// TIA Portal project "Project_teste" (V17)

(* hardware
DEVICE "S7-1200 station_1"  S7-1200 Station
   slot 0: "Rack_0"  S7-1200 Rack  Rack  V1.0
   slot 1: "PLC_1"  CPU 1214C DC/DC/DC  6ES7 214-1AG40-0XB0  V4.4
*)

// ===== PLC "PLC_1"  CPU 1214C DC/DC/DC =====

VAR_GLOBAL   // PLC tag table "Default tag table"
   "liga" AT %I0.0 : Bool;
   "velocidade" AT %MW2 : UInt;
   "velocidade_motor" AT %MW4 : Word;
   "corrente_motor" AT %MW6 : Word;
   "falha_motor" AT %MW8 : Word;
   "troca_ref" AT %I0.1 : Bool;
END_VAR

TYPE "driver_config"
   STRUCT
      MB_client : TCON_IP_v4;
   END_STRUCT;
   // MB_client.InterfaceId := 64;
   // MB_client.ID := 1;
   // MB_client.ConnectionType := 11;
   // MB_client.ActiveEstablished := true;
   // MB_client.RemotePort := 502;
   // MB_client.LocalPort := 502;
END_TYPE

TYPE "driver_comunic"
   STRUCT
      parametros : Array[0..3] of UDInt;
      leitura_escrita : Array[0..3] of Bool;
      dado_leitura : Array[0..3] of Word;
      dado_escrita : Array[0..3] of Word;
      trigger : Array[0..3] of Bool;
   END_STRUCT;
END_TYPE

DATA_BLOCK "configuracao"   // DB1
{ S7_Optimized_Access := 'TRUE' }
VERSION : 0.1
BEGIN
   MB_client.RemoteAddress.ADDR[1] := 172;
   MB_client.RemoteAddress.ADDR[2] := 16;
   MB_client.RemoteAddress.ADDR[3] := 80;
   MB_client.RemoteAddress.ADDR[4] := 30;
END_DATA_BLOCK

DATA_BLOCK "comunicacao"   // DB2
{ S7_Optimized_Access := 'TRUE' }
VERSION : 0.1
BEGIN
END_DATA_BLOCK

DATA_BLOCK "Driver_CFW500_DB"   // DB4
{ S7_Optimized_Access := 'TRUE' }
VERSION : 0.1
// stored: InstanceOfName Driver_CFW500
"Driver_CFW500"
BEGIN
END_DATA_BLOCK

FUNCTION_BLOCK "transicao_estados"   // FB1, SCL
{ S7_Optimized_Access := 'FALSE' }
VERSION : 0.1
   VAR_INPUT
      liga : Bool;
      ref_velocidade : UInt;
      rampa_aceleracao : UInt;
      rampa_desaceleracao : UInt;
   END_VAR
BEGIN
   CASE "Driver_CFW500_DB".estado OF
       0:
           IF NOT "Driver_CFW500_DB".saidas_atualizadas THEN
               "Driver_CFW500_DB".estado := 1;
           END_IF;
       1:
           IF "Driver_CFW500_DB".saidas_atualizadas THEN
               "Driver_CFW500_DB".estado := 10;
           END_IF;
       10:  
           IF #liga <> "Driver_CFW500_DB".ligar_old THEN
               "Driver_CFW500_DB".estado := 100;
           ELSE
               "Driver_CFW500_DB".estado := 11;
           END_IF;
       11:  
           IF #ref_velocidade <> "Driver_CFW500_DB".ref_velocidade_old THEN
               "Driver_CFW500_DB".estado := 101;
           ELSE
               "Driver_CFW500_DB".estado := 12;
           END_IF;
       12:
           IF #rampa_aceleracao <> "Driver_CFW500_DB".rampa_aceleracao_old THEN
               "Driver_CFW500_DB".estado := 102;
           ELSE
               "Driver_CFW500_DB".estado := 13;
           END_IF;
       13:
           IF #rampa_desaceleracao <> "Driver_CFW500_DB".rampa_desaceleracao_old THEN
               "Driver_CFW500_DB".estado := 103;
           ELSE
               "Driver_CFW500_DB".estado := 49;
           END_IF;
       49:
           IF NOT "Driver_CFW500_DB".param_var_atualizados THEN
               "Driver_CFW500_DB".estado := 50;
           END_IF;
       50:
           IF "Driver_CFW500_DB".param_var_atualizados THEN
               "Driver_CFW500_DB".estado := 0;
           END_IF;
       100:
           IF #liga = "Driver_CFW500_DB".ligar_old THEN
               "Driver_CFW500_DB".estado := 49;
           END_IF;
       101:
           IF #ref_velocidade = "Driver_CFW500_DB".ref_velocidade_old THEN
               "Driver_CFW500_DB".estado := 49;
           END_IF;
       102:
           IF #rampa_aceleracao = "Driver_CFW500_DB".rampa_aceleracao_old THEN
               "Driver_CFW500_DB".estado := 49;
           END_IF;
       103:
           IF #rampa_desaceleracao = "Driver_CFW500_DB".rampa_desaceleracao_old THEN
               "Driver_CFW500_DB".estado := 49;
           END_IF;
   END_CASE;
END_FUNCTION_BLOCK

FUNCTION_BLOCK "escrever_parametro"   // FB2, SCL
{ S7_Optimized_Access := 'FALSE' }
VERSION : 0.1
   VAR_INPUT
      parametro : UDInt;
      dado : Word;
      escrever : Bool;
   END_VAR
   VAR_OUTPUT
      escrito : Bool;
   END_VAR
   VAR
      flag_start : Bool;
   END_VAR
BEGIN
   IF #escrever AND
      NOT #flag_start AND
      NOT "Driver_CFW500_DB".disconnect AND
      NOT "Driver_CFW500_DB".busy THEN

       #escrito := 0;

       // Define modo de escrita
       "Driver_CFW500_DB".mode := 1;

       // Define comprimento da escrita
       "Driver_CFW500_DB".data_len := 1;

       // Define endereço para escrita
       "Driver_CFW500_DB".data_addr := #parametro + 40001;

       // Define dado para escrita
       "Driver_CFW500_DB".data_ptr[0] := #dado;

       // Gera pulso para disparar requisição de escrita
       "Driver_CFW500_DB".req := 1;

       #flag_start := TRUE;

   ELSIF #flag_start AND "Driver_CFW500_DB".busy THEN
       "Driver_CFW500_DB".req := FALSE;

   ELSIF #flag_start AND
      ("Driver_CFW500_DB".done OR "Driver_CFW500_DB".error) THEN
      #flag_start := FALSE;
      #escrito := TRUE;

   END_IF;
END_FUNCTION_BLOCK

FUNCTION_BLOCK "ler_parametro"   // FB3, SCL
{ S7_Optimized_Access := 'FALSE' }
VERSION : 0.1
   VAR_INPUT
      parametro : UDInt;
      ler : Bool;
   END_VAR
   VAR_OUTPUT
      dado : Word;
      lido : Bool;
   END_VAR
   VAR
      flag_start : Bool;
   END_VAR
BEGIN
   IF #ler AND
       NOT #flag_start AND
       NOT "Driver_CFW500_DB".disconnect AND
       NOT "Driver_CFW500_DB".busy THEN

       //    "Driver_CFW500_DB".data_ptr[0] := 0;
       //    #dado := 0;
       #lido := FALSE;

       // Define modo de leitura
       "Driver_CFW500_DB".mode := 0;

       // Define comprimento da leitura
       "Driver_CFW500_DB".data_len := 1;

       // Define endereço para leitura
       "Driver_CFW500_DB".data_addr := #parametro + 40001;

       // Gera pulso para disparar requisição de leitura
       "Driver_CFW500_DB".req := 1;

       #flag_start := TRUE;

   ELSIF #flag_start AND "Driver_CFW500_DB".busy THEN
       "Driver_CFW500_DB".req := FALSE;

   ELSIF #flag_start AND
         NOT "Driver_CFW500_DB".req AND
         ("Driver_CFW500_DB".done OR "Driver_CFW500_DB".error) THEN

       #flag_start := FALSE;
       #dado := "Driver_CFW500_DB".data_ptr[0];
       #lido := TRUE;

   END_IF;
END_FUNCTION_BLOCK

FUNCTION_BLOCK "acoes_estado"   // FB4, LAD
{ S7_Optimized_Access := 'FALSE' }
VERSION : 0.1
   VAR_INPUT
      ligar : Bool;
      ref_vel : Word;
      rampa_acel : Word;
      rampa_desacel : Word;
   END_VAR
   VAR_OUTPUT
      velocidade : Word;
      corrente : Word;
      falha : Word;
   END_VAR
   VAR
      aux0 : Bool;
      aux1 : Bool;
      aux2 : Bool;
      aux3 : Bool;
      aux4 : Bool;
      aux5 : Bool;
      aux6 : Bool;
      aux7 : Bool;
      aux10 : Bool;
      aux11 : Bool;
      aux12 : Bool;
      aux13 : Bool;
      aux20 : Bool;
      aux21 : Bool;
      aux22 : Bool;
      aux23 : Bool;
      aux30 : Bool;
      aux31 : Bool;
      aux32 : Bool;
      aux33 : Bool;
      aux100 : Bool;
      aux101 : Bool;
      aux102 : Bool;
      aux103 : Bool;
      aux104 : Bool;
      aux105 : Bool;
      aux106 : Bool;
      aux107 : Bool;
      aux200 : Bool;
      aux201 : Bool;
      aux202 : Bool;
      aux203 : Bool;
      aux204 : Bool;
      aux205 : Bool;
      aux206 : Bool;
      aux207 : Bool;
      aux208 : Bool;
      aux209 : Bool;
      aux210 : Bool;
      aux211 : Bool;
      atualizar_p0 : Bool;
      atualizar_p1 : Bool;
      atualizar_p2 : Bool;
      atualizar_p3 : Bool;
      ler_vel : "ler_parametro";
      ler_cor : "ler_parametro";
      ler_falha : "ler_parametro";
      escrever_liga : "escrever_parametro";
      escrever_desliga : "escrever_parametro";
      escrever_ref : "escrever_parametro";
      escrever_acel : "escrever_parametro";
      escrever_desacel : "escrever_parametro";
      est_50 : "estado 50";
      temporiza : IEC_TIMER;
   END_VAR
   VAR_TEMP   // added for the SCL form of the ladder/FBD networks
      _w1 : Bool;
      _w2 : Bool;
      _w3 : Bool;
      _w4 : Bool;
      _w5 : Bool;
   END_VAR
BEGIN

REGION Network 1: Estado 0
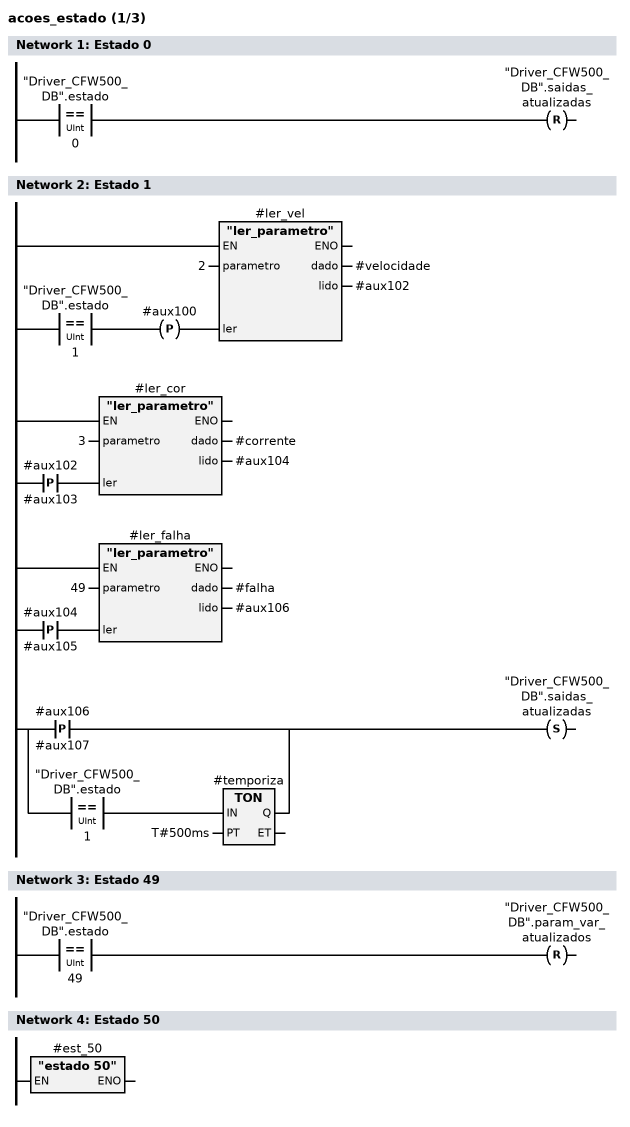
   RUNG wire#powerrail
      { S7_Templates := "SrcType := UInt" } EQ_Contact(in1 := "Driver_CFW500_DB".estado, in2 := 0)
      R_Coil( "Driver_CFW500_DB".saidas_atualizadas )
   END_RUNG
   // the same network as SCL:
   IF "Driver_CFW500_DB".estado = 0 THEN "Driver_CFW500_DB".saidas_atualizadas := FALSE; END_IF;
END_REGION

REGION Network 2: Estado 1
   #_w1 := "Driver_CFW500_DB".estado = 1;
   #_w2 := #_w1 AND NOT #aux100;   // rising edge
   #aux100 := #_w1;
   #ler_vel(parametro := 2, ler := #_w2, dado => #velocidade, lido => #aux102);   // "ler_parametro"
   #_w3 := #aux102 AND NOT #aux103;   // rising edge of #aux102
   #aux103 := #aux102;
   #ler_cor(parametro := 3, ler := #_w3, dado => #corrente, lido => #aux104);   // "ler_parametro"
   #_w4 := #aux104 AND NOT #aux105;   // rising edge of #aux104
   #aux105 := #aux104;
   #ler_falha(parametro := 49, ler := #_w4, dado => #falha, lido => #aux106);   // "ler_parametro"
   #_w5 := #aux106 AND NOT #aux107;   // rising edge of #aux106
   #aux107 := #aux106;
   #temporiza.TON(IN := "Driver_CFW500_DB".estado = 1, PT := T#500ms);
   IF #_w5 OR #temporiza.Q THEN "Driver_CFW500_DB".saidas_atualizadas := TRUE; END_IF;
END_REGION

REGION Network 3: Estado 49
   RUNG wire#powerrail
      { S7_Templates := "SrcType := UInt" } EQ_Contact(in1 := "Driver_CFW500_DB".estado, in2 := 49)
      R_Coil( "Driver_CFW500_DB".param_var_atualizados )
   END_RUNG
   // the same network as SCL:
   IF "Driver_CFW500_DB".estado = 49 THEN "Driver_CFW500_DB".param_var_atualizados := FALSE; END_IF;
END_REGION

REGION Network 4: Estado 50
   RUNG wire#powerrail
      #est_50()
   END_RUNG
   // the same network as SCL:
   #est_50();   // "estado 50"
END_REGION

REGION Network 5: Estado 100
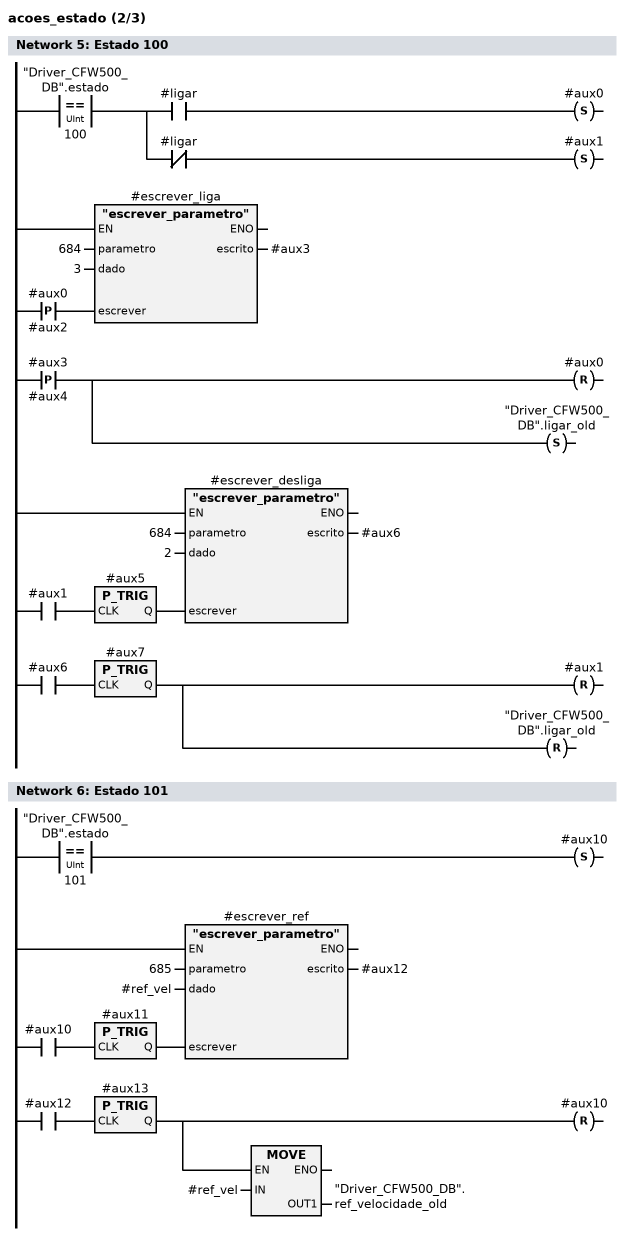
   RUNG wire#powerrail
      { S7_Templates := "SrcType := UInt" } EQ_Contact(in1 := "Driver_CFW500_DB".estado, in2 := 100)
      wire#w1
      Contact( #ligar )
      S_Coil( #aux0 )
   END_RUNG
   RUNG wire#w1
      I_Contact( #ligar )
      S_Coil( #aux1 )
   END_RUNG
   RUNG wire#powerrail
      #escrever_liga(escrever := wire#w2, parametro := 684, dado := 3, escrito => #aux3)
   END_RUNG
   RUNG wire#powerrail
      P_Contact(operand := #aux0, bit := #aux2)
   END_RUNG wire#w2
   RUNG wire#powerrail
      P_Contact(operand := #aux3, bit := #aux4)
      wire#w3
      R_Coil( #aux0 )
   END_RUNG
   RUNG wire#w3
      S_Coil( "Driver_CFW500_DB".ligar_old )
   END_RUNG
   RUNG wire#powerrail
      #escrever_desliga(escrever := wire#w4, parametro := 684, dado := 2, escrito => #aux6)
   END_RUNG
   RUNG wire#powerrail
      Contact( #aux1 )
      P_Trig( #aux5 )
   END_RUNG wire#w4
   RUNG wire#powerrail
      Contact( #aux6 )
      P_Trig( #aux7 )
      wire#w5
      R_Coil( #aux1 )
   END_RUNG
   RUNG wire#w5
      R_Coil( "Driver_CFW500_DB".ligar_old )
   END_RUNG
   // the same network as SCL:
   #_w1 := "Driver_CFW500_DB".estado = 100;
   IF #_w1 AND #ligar THEN #aux0 := TRUE; END_IF;
   IF #_w1 AND NOT #ligar THEN #aux1 := TRUE; END_IF;
   #_w2 := #aux0 AND NOT #aux2;   // rising edge of #aux0
   #aux2 := #aux0;
   #escrever_liga(parametro := 684, dado := 3, escrever := #_w2, escrito => #aux3);   // "escrever_parametro"
   #_w3 := #aux3 AND NOT #aux4;   // rising edge of #aux3
   #aux4 := #aux3;
   IF #_w3 THEN
       #aux0 := FALSE;
       "Driver_CFW500_DB".ligar_old := TRUE;
   END_IF;
   #_w4 := #aux1 AND NOT #aux5;   // rising edge
   #aux5 := #aux1;
   #escrever_desliga(parametro := 684, dado := 2, escrever := #_w4, escrito => #aux6);   // "escrever_parametro"
   #_w5 := #aux6 AND NOT #aux7;   // rising edge
   #aux7 := #aux6;
   IF #_w5 THEN
       #aux1 := FALSE;
       "Driver_CFW500_DB".ligar_old := FALSE;
   END_IF;
END_REGION

REGION Network 6: Estado 101
   RUNG wire#powerrail
      { S7_Templates := "SrcType := UInt" } EQ_Contact(in1 := "Driver_CFW500_DB".estado, in2 := 101)
      S_Coil( #aux10 )
   END_RUNG
   RUNG wire#powerrail
      #escrever_ref(escrever := wire#w1, parametro := 685, dado := #ref_vel, escrito => #aux12)
   END_RUNG
   RUNG wire#powerrail
      Contact( #aux10 )
      P_Trig( #aux11 )
   END_RUNG wire#w1
   RUNG wire#powerrail
      Contact( #aux12 )
      P_Trig( #aux13 )
      wire#w2
      R_Coil( #aux10 )
   END_RUNG
   RUNG wire#w2
      Move(in := #ref_vel, out1 => "Driver_CFW500_DB".ref_velocidade_old)
   END_RUNG
   // the same network as SCL:
   IF "Driver_CFW500_DB".estado = 101 THEN #aux10 := TRUE; END_IF;
   #_w1 := #aux10 AND NOT #aux11;   // rising edge
   #aux11 := #aux10;
   #escrever_ref(parametro := 685, dado := #ref_vel, escrever := #_w1, escrito => #aux12);   // "escrever_parametro"
   #_w2 := #aux12 AND NOT #aux13;   // rising edge
   #aux13 := #aux12;
   IF #_w2 THEN
       #aux10 := FALSE;
       "Driver_CFW500_DB".ref_velocidade_old := #ref_vel;
   END_IF;
END_REGION

REGION Network 7: Estado 102
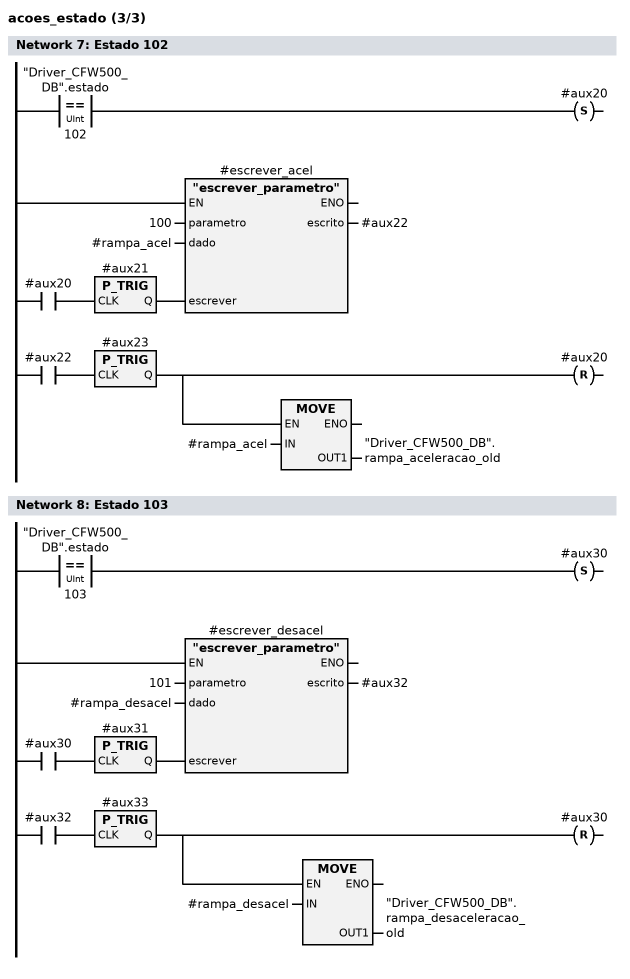
   RUNG wire#powerrail
      { S7_Templates := "SrcType := UInt" } EQ_Contact(in1 := "Driver_CFW500_DB".estado, in2 := 102)
      S_Coil( #aux20 )
   END_RUNG
   RUNG wire#powerrail
      #escrever_acel(escrever := wire#w1, parametro := 100, dado := #rampa_acel, escrito => #aux22)
   END_RUNG
   RUNG wire#powerrail
      Contact( #aux20 )
      P_Trig( #aux21 )
   END_RUNG wire#w1
   RUNG wire#powerrail
      Contact( #aux22 )
      P_Trig( #aux23 )
      wire#w2
      R_Coil( #aux20 )
   END_RUNG
   RUNG wire#w2
      Move(in := #rampa_acel, out1 => "Driver_CFW500_DB".rampa_aceleracao_old)
   END_RUNG
   // the same network as SCL:
   IF "Driver_CFW500_DB".estado = 102 THEN #aux20 := TRUE; END_IF;
   #_w1 := #aux20 AND NOT #aux21;   // rising edge
   #aux21 := #aux20;
   #escrever_acel(parametro := 100, dado := #rampa_acel, escrever := #_w1, escrito => #aux22);   // "escrever_parametro"
   #_w2 := #aux22 AND NOT #aux23;   // rising edge
   #aux23 := #aux22;
   IF #_w2 THEN
       #aux20 := FALSE;
       "Driver_CFW500_DB".rampa_aceleracao_old := #rampa_acel;
   END_IF;
END_REGION

REGION Network 8: Estado 103
   RUNG wire#powerrail
      { S7_Templates := "SrcType := UInt" } EQ_Contact(in1 := "Driver_CFW500_DB".estado, in2 := 103)
      S_Coil( #aux30 )
   END_RUNG
   RUNG wire#powerrail
      #escrever_desacel(escrever := wire#w1, parametro := 101, dado := #rampa_desacel, escrito => #aux32)
   END_RUNG
   RUNG wire#powerrail
      Contact( #aux30 )
      P_Trig( #aux31 )
   END_RUNG wire#w1
   RUNG wire#powerrail
      Contact( #aux32 )
      P_Trig( #aux33 )
      wire#w2
      R_Coil( #aux30 )
   END_RUNG
   RUNG wire#w2
      Move(in := #rampa_desacel, out1 => "Driver_CFW500_DB".rampa_desaceleracao_old)
   END_RUNG
   // the same network as SCL:
   IF "Driver_CFW500_DB".estado = 103 THEN #aux30 := TRUE; END_IF;
   #_w1 := #aux30 AND NOT #aux31;   // rising edge
   #aux31 := #aux30;
   #escrever_desacel(parametro := 101, dado := #rampa_desacel, escrever := #_w1, escrito => #aux32);   // "escrever_parametro"
   #_w2 := #aux32 AND NOT #aux33;   // rising edge
   #aux33 := #aux32;
   IF #_w2 THEN
       #aux30 := FALSE;
       "Driver_CFW500_DB".rampa_desaceleracao_old := #rampa_desacel;
   END_IF;
END_REGION
END_FUNCTION_BLOCK

FUNCTION_BLOCK "Driver_CFW500"   // FB5, LAD
{ S7_Optimized_Access := 'TRUE' }
VERSION : 0.1
   VAR_INPUT
      ligar : Bool;
      ref_velocidade : UInt;
      rampa_aceleracao : UInt;
      rampa_desaceleracao : UInt;
   END_VAR
   VAR_OUTPUT
      velocidade : Word;
      corrente : Word;
      falha : Word;
   END_VAR
   VAR_IN_OUT
      config : "driver_config";
      comunic : "driver_comunic";
   END_VAR
   VAR
      mb_client_db : MB_CLIENT;
      acoes : "acoes_estado";
      transicoes : "transicao_estados";
      req : Bool;
      disconnect : Bool;
      mode : USInt;
      data_addr : UDInt;
      data_len : UInt;
      data_ptr : Array[0..9] of Word;
      done : Bool;
      busy : Bool;
      error : Bool;
      status : Word;
      estado : UInt;
      dado_p684 : Word;
      ligar_old : Bool;
      ref_velocidade_old : UInt;
      rampa_aceleracao_old : UInt;
      rampa_desaceleracao_old : UInt;
      "dados[0]_old" : Word;
      "dados[1]_old" : Word;
      "dados[2]_old" : Word;
      "dados[3]_old" : Word;
      saidas_atualizadas : Bool;
      param_var_atualizados : Bool;
   END_VAR
BEGIN

REGION Network 1
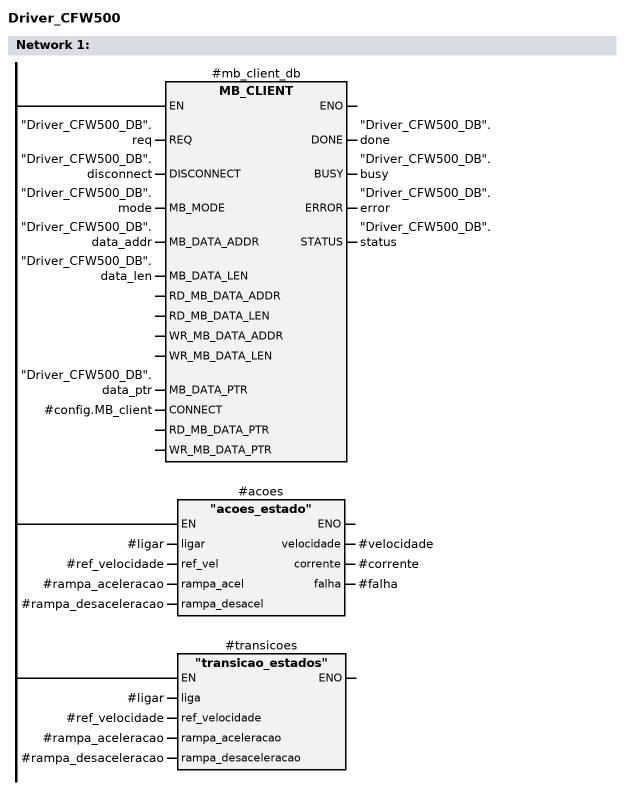
   #mb_client_db(REQ := "Driver_CFW500_DB".req,   // MB_CLIENT
                 DISCONNECT := "Driver_CFW500_DB".disconnect,
                 MB_MODE := "Driver_CFW500_DB".mode,
                 MB_DATA_ADDR := "Driver_CFW500_DB".data_addr,
                 MB_DATA_LEN := "Driver_CFW500_DB".data_len,
                 MB_DATA_PTR := "Driver_CFW500_DB".data_ptr,
                 CONNECT := #config.MB_client,
                 DONE => "Driver_CFW500_DB".done,
                 BUSY => "Driver_CFW500_DB".busy,
                 ERROR => "Driver_CFW500_DB".error,
                 STATUS => "Driver_CFW500_DB".status);
   #acoes(ligar := #ligar,   // "acoes_estado"
          ref_vel := #ref_velocidade,
          rampa_acel := #rampa_aceleracao,
          rampa_desacel := #rampa_desaceleracao,
          velocidade => #velocidade,
          corrente => #corrente,
          falha => #falha);
   #transicoes(liga := #ligar,   // "transicao_estados"
               ref_velocidade := #ref_velocidade,
               rampa_aceleracao := #rampa_aceleracao,
               rampa_desaceleracao := #rampa_desaceleracao);
END_REGION
END_FUNCTION_BLOCK

FUNCTION_BLOCK "estado 50"   // FB6, LAD
{ S7_Optimized_Access := 'TRUE' }
VERSION : 0.1
   VAR
      p_1 : Bool;
      aux1 : Bool;
      aux2 : Bool;
      aux3 : Bool;
      aux4 : Bool;
      aux5 : Bool;
      aux6 : Bool;
      aux7 : Bool;
      p_2 : Bool;
      ler_1 : "ler_parametro";
      ler_2 : "ler_parametro";
      ler_3 : "ler_parametro";
      ler_4 : "ler_parametro";
      escrever_1 : "escrever_parametro";
      escrever_2 : "escrever_parametro";
      escrever_3 : "escrever_parametro";
      escrever_4 : "escrever_parametro";
      aux10 : Bool;
      aux11 : Bool;
      aux12 : Bool;
      aux13 : Bool;
      aux14 : Bool;
      aux15 : Bool;
      p_3 : Bool;
      aux20 : Bool;
      aux21 : Bool;
      aux22 : Bool;
      aux23 : Bool;
      aux24 : Bool;
      aux25 : Bool;
      p_4 : Bool;
      aux30 : Bool;
      aux31 : Bool;
      aux32 : Bool;
      aux33 : Bool;
      aux34 : Bool;
      aux35 : Bool;
      aux0 : Bool;
   END_VAR
   VAR_TEMP   // added for the SCL form of the ladder/FBD networks
      _w1 : Bool;
      _w2 : Bool;
      _w3 : Bool;
      _w4 : Bool;
      _w5 : Bool;
      _w6 : Bool;
      _w7 : Bool;
      _w8 : Bool;
   END_VAR
BEGIN

REGION Network 1
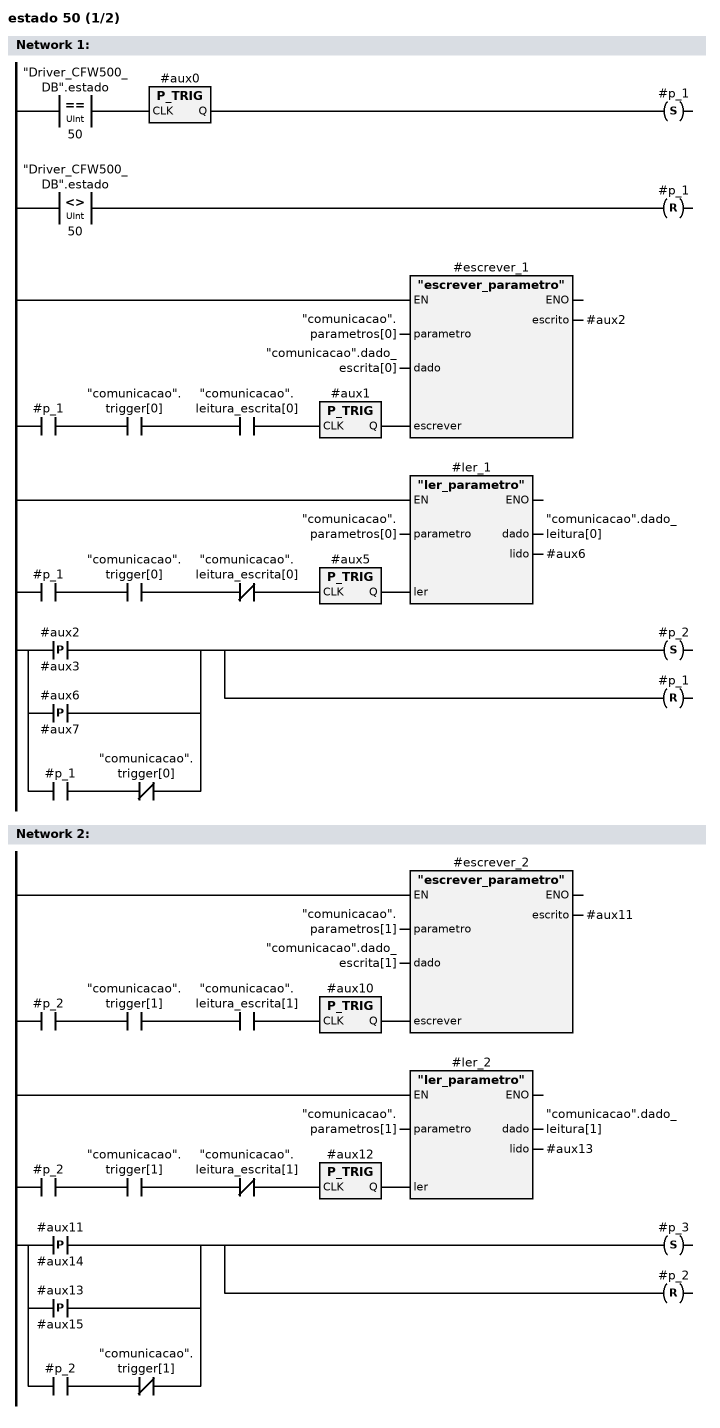
   RUNG wire#powerrail
      { S7_Templates := "SrcType := UInt" } EQ_Contact(in1 := "Driver_CFW500_DB".estado, in2 := 50)
      P_Trig( #aux0 )
      S_Coil( #p_1 )
   END_RUNG
   RUNG wire#powerrail
      { S7_Templates := "SrcType := UInt" } NE_Contact(in1 := "Driver_CFW500_DB".estado, in2 := 50)
      R_Coil( #p_1 )
   END_RUNG
   RUNG wire#powerrail
      #escrever_1(escrever := wire#w1, parametro := "comunicacao".parametros[0], dado := "comunicacao".dado_escrita[0], escrito => #aux2)
   END_RUNG
   RUNG wire#powerrail
      Contact( #p_1 )
      Contact( "comunicacao".trigger[0] )
      Contact( "comunicacao".leitura_escrita[0] )
      P_Trig( #aux1 )
   END_RUNG wire#w1
   RUNG wire#powerrail
      #ler_1(ler := wire#w2, parametro := "comunicacao".parametros[0], dado => "comunicacao".dado_leitura[0], lido => #aux6)
   END_RUNG
   RUNG wire#powerrail
      Contact( #p_1 )
      Contact( "comunicacao".trigger[0] )
      I_Contact( "comunicacao".leitura_escrita[0] )
      P_Trig( #aux5 )
   END_RUNG wire#w2
   RUNG wire#powerrail
      P_Contact(operand := #aux2, bit := #aux3)
      wire#w3
      S_Coil( #p_2 )
   END_RUNG
   RUNG wire#powerrail
      P_Contact(operand := #aux6, bit := #aux7)
   END_RUNG wire#w3
   RUNG wire#powerrail
      Contact( #p_1 )
      I_Contact( "comunicacao".trigger[0] )
   END_RUNG wire#w3
   RUNG wire#w3
      R_Coil( #p_1 )
   END_RUNG
   // the same network as SCL:
   #_w1 := "Driver_CFW500_DB".estado = 50;
   #_w2 := #_w1 AND NOT #aux0;   // rising edge
   #aux0 := #_w1;
   IF #_w2 THEN #p_1 := TRUE; END_IF;
   IF "Driver_CFW500_DB".estado <> 50 THEN #p_1 := FALSE; END_IF;
   #_w3 := #p_1 AND "comunicacao".trigger[0] AND "comunicacao".leitura_escrita[0];
   #_w4 := #_w3 AND NOT #aux1;   // rising edge
   #aux1 := #_w3;
   #escrever_1(parametro := "comunicacao".parametros[0],   // "escrever_parametro"
               dado := "comunicacao".dado_escrita[0],
               escrever := #_w4,
               escrito => #aux2);
   #_w5 := #p_1 AND "comunicacao".trigger[0] AND NOT "comunicacao".leitura_escrita[0];
   #_w6 := #_w5 AND NOT #aux5;   // rising edge
   #aux5 := #_w5;
   #ler_1(parametro := "comunicacao".parametros[0],   // "ler_parametro"
          ler := #_w6,
          dado => "comunicacao".dado_leitura[0],
          lido => #aux6);
   #_w7 := #aux2 AND NOT #aux3;   // rising edge of #aux2
   #aux3 := #aux2;
   #_w8 := #aux6 AND NOT #aux7;   // rising edge of #aux6
   #aux7 := #aux6;
   IF #_w7 OR #_w8 OR (#p_1 AND NOT "comunicacao".trigger[0]) THEN
       #p_2 := TRUE;
       #p_1 := FALSE;
   END_IF;
END_REGION

REGION Network 2
   RUNG wire#powerrail
      #escrever_2(escrever := wire#w1, parametro := "comunicacao".parametros[1], dado := "comunicacao".dado_escrita[1], escrito => #aux11)
   END_RUNG
   RUNG wire#powerrail
      Contact( #p_2 )
      Contact( "comunicacao".trigger[1] )
      Contact( "comunicacao".leitura_escrita[1] )
      P_Trig( #aux10 )
   END_RUNG wire#w1
   RUNG wire#powerrail
      #ler_2(ler := wire#w2, parametro := "comunicacao".parametros[1], dado => "comunicacao".dado_leitura[1], lido => #aux13)
   END_RUNG
   RUNG wire#powerrail
      Contact( #p_2 )
      Contact( "comunicacao".trigger[1] )
      I_Contact( "comunicacao".leitura_escrita[1] )
      P_Trig( #aux12 )
   END_RUNG wire#w2
   RUNG wire#powerrail
      P_Contact(operand := #aux11, bit := #aux14)
      wire#w3
      S_Coil( #p_3 )
   END_RUNG
   RUNG wire#powerrail
      P_Contact(operand := #aux13, bit := #aux15)
   END_RUNG wire#w3
   RUNG wire#powerrail
      Contact( #p_2 )
      I_Contact( "comunicacao".trigger[1] )
   END_RUNG wire#w3
   RUNG wire#w3
      R_Coil( #p_2 )
   END_RUNG
   // the same network as SCL:
   #_w1 := #p_2 AND "comunicacao".trigger[1] AND "comunicacao".leitura_escrita[1];
   #_w2 := #_w1 AND NOT #aux10;   // rising edge
   #aux10 := #_w1;
   #escrever_2(parametro := "comunicacao".parametros[1],   // "escrever_parametro"
               dado := "comunicacao".dado_escrita[1],
               escrever := #_w2,
               escrito => #aux11);
   #_w3 := #p_2 AND "comunicacao".trigger[1] AND NOT "comunicacao".leitura_escrita[1];
   #_w4 := #_w3 AND NOT #aux12;   // rising edge
   #aux12 := #_w3;
   #ler_2(parametro := "comunicacao".parametros[1],   // "ler_parametro"
          ler := #_w4,
          dado => "comunicacao".dado_leitura[1],
          lido => #aux13);
   #_w5 := #aux11 AND NOT #aux14;   // rising edge of #aux11
   #aux14 := #aux11;
   #_w6 := #aux13 AND NOT #aux15;   // rising edge of #aux13
   #aux15 := #aux13;
   IF #_w5 OR #_w6 OR (#p_2 AND NOT "comunicacao".trigger[1]) THEN
       #p_3 := TRUE;
       #p_2 := FALSE;
   END_IF;
END_REGION

REGION Network 3
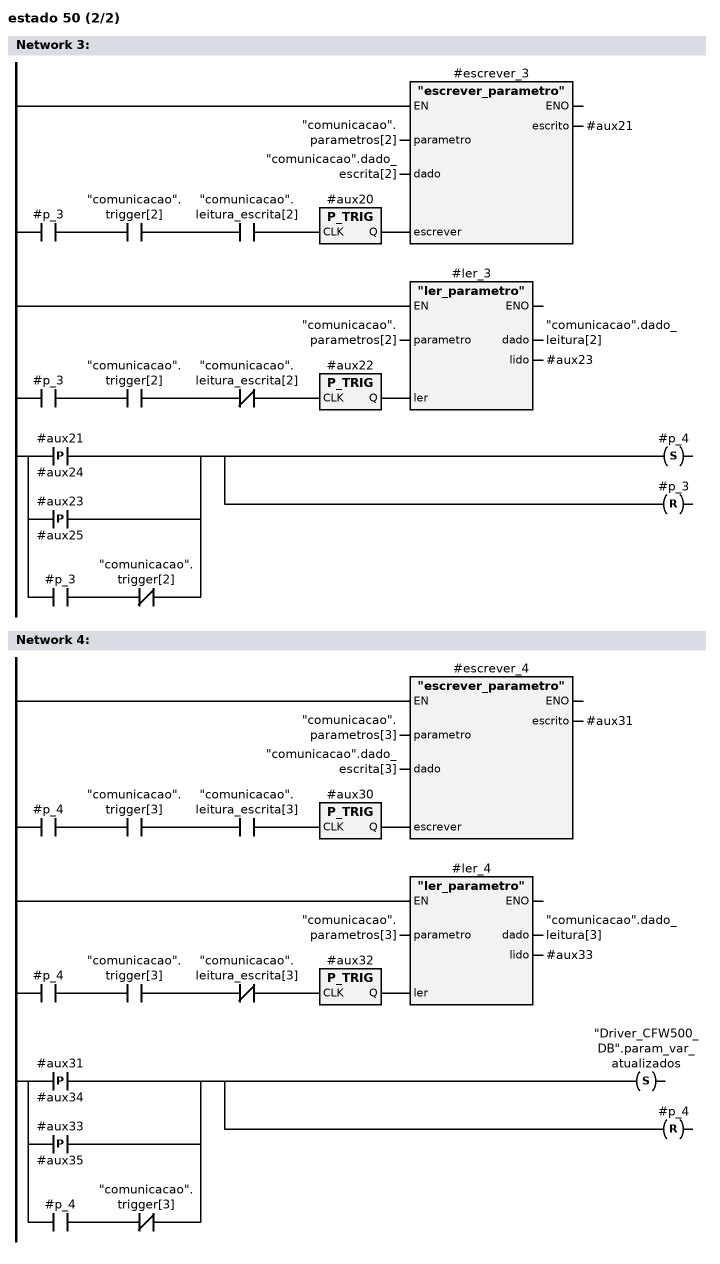
   RUNG wire#powerrail
      #escrever_3(escrever := wire#w1, parametro := "comunicacao".parametros[2], dado := "comunicacao".dado_escrita[2], escrito => #aux21)
   END_RUNG
   RUNG wire#powerrail
      Contact( #p_3 )
      Contact( "comunicacao".trigger[2] )
      Contact( "comunicacao".leitura_escrita[2] )
      P_Trig( #aux20 )
   END_RUNG wire#w1
   RUNG wire#powerrail
      #ler_3(ler := wire#w2, parametro := "comunicacao".parametros[2], dado => "comunicacao".dado_leitura[2], lido => #aux23)
   END_RUNG
   RUNG wire#powerrail
      Contact( #p_3 )
      Contact( "comunicacao".trigger[2] )
      I_Contact( "comunicacao".leitura_escrita[2] )
      P_Trig( #aux22 )
   END_RUNG wire#w2
   RUNG wire#powerrail
      P_Contact(operand := #aux21, bit := #aux24)
      wire#w3
      S_Coil( #p_4 )
   END_RUNG
   RUNG wire#powerrail
      P_Contact(operand := #aux23, bit := #aux25)
   END_RUNG wire#w3
   RUNG wire#powerrail
      Contact( #p_3 )
      I_Contact( "comunicacao".trigger[2] )
   END_RUNG wire#w3
   RUNG wire#w3
      R_Coil( #p_3 )
   END_RUNG
   // the same network as SCL:
   #_w1 := #p_3 AND "comunicacao".trigger[2] AND "comunicacao".leitura_escrita[2];
   #_w2 := #_w1 AND NOT #aux20;   // rising edge
   #aux20 := #_w1;
   #escrever_3(parametro := "comunicacao".parametros[2],   // "escrever_parametro"
               dado := "comunicacao".dado_escrita[2],
               escrever := #_w2,
               escrito => #aux21);
   #_w3 := #p_3 AND "comunicacao".trigger[2] AND NOT "comunicacao".leitura_escrita[2];
   #_w4 := #_w3 AND NOT #aux22;   // rising edge
   #aux22 := #_w3;
   #ler_3(parametro := "comunicacao".parametros[2],   // "ler_parametro"
          ler := #_w4,
          dado => "comunicacao".dado_leitura[2],
          lido => #aux23);
   #_w5 := #aux21 AND NOT #aux24;   // rising edge of #aux21
   #aux24 := #aux21;
   #_w6 := #aux23 AND NOT #aux25;   // rising edge of #aux23
   #aux25 := #aux23;
   IF #_w5 OR #_w6 OR (#p_3 AND NOT "comunicacao".trigger[2]) THEN
       #p_4 := TRUE;
       #p_3 := FALSE;
   END_IF;
END_REGION

REGION Network 4
   RUNG wire#powerrail
      #escrever_4(escrever := wire#w1, parametro := "comunicacao".parametros[3], dado := "comunicacao".dado_escrita[3], escrito => #aux31)
   END_RUNG
   RUNG wire#powerrail
      Contact( #p_4 )
      Contact( "comunicacao".trigger[3] )
      Contact( "comunicacao".leitura_escrita[3] )
      P_Trig( #aux30 )
   END_RUNG wire#w1
   RUNG wire#powerrail
      #ler_4(ler := wire#w2, parametro := "comunicacao".parametros[3], dado => "comunicacao".dado_leitura[3], lido => #aux33)
   END_RUNG
   RUNG wire#powerrail
      Contact( #p_4 )
      Contact( "comunicacao".trigger[3] )
      I_Contact( "comunicacao".leitura_escrita[3] )
      P_Trig( #aux32 )
   END_RUNG wire#w2
   RUNG wire#powerrail
      P_Contact(operand := #aux31, bit := #aux34)
      wire#w3
      S_Coil( "Driver_CFW500_DB".param_var_atualizados )
   END_RUNG
   RUNG wire#powerrail
      P_Contact(operand := #aux33, bit := #aux35)
   END_RUNG wire#w3
   RUNG wire#powerrail
      Contact( #p_4 )
      I_Contact( "comunicacao".trigger[3] )
   END_RUNG wire#w3
   RUNG wire#w3
      R_Coil( #p_4 )
   END_RUNG
   // the same network as SCL:
   #_w1 := #p_4 AND "comunicacao".trigger[3] AND "comunicacao".leitura_escrita[3];
   #_w2 := #_w1 AND NOT #aux30;   // rising edge
   #aux30 := #_w1;
   #escrever_4(parametro := "comunicacao".parametros[3],   // "escrever_parametro"
               dado := "comunicacao".dado_escrita[3],
               escrever := #_w2,
               escrito => #aux31);
   #_w3 := #p_4 AND "comunicacao".trigger[3] AND NOT "comunicacao".leitura_escrita[3];
   #_w4 := #_w3 AND NOT #aux32;   // rising edge
   #aux32 := #_w3;
   #ler_4(parametro := "comunicacao".parametros[3],   // "ler_parametro"
          ler := #_w4,
          dado => "comunicacao".dado_leitura[3],
          lido => #aux33);
   #_w5 := #aux31 AND NOT #aux34;   // rising edge of #aux31
   #aux34 := #aux31;
   #_w6 := #aux33 AND NOT #aux35;   // rising edge of #aux33
   #aux35 := #aux33;
   IF #_w5 OR #_w6 OR (#p_4 AND NOT "comunicacao".trigger[3]) THEN
       "Driver_CFW500_DB".param_var_atualizados := TRUE;
       #p_4 := FALSE;
   END_IF;
END_REGION
END_FUNCTION_BLOCK

ORGANIZATION_BLOCK "Main"   // OB1, LAD, ProgramCycle
TITLE = "Main Program Sweep (Cycle)"
{ S7_Optimized_Access := 'TRUE' }
VERSION : 0.1
   VAR_INPUT
      Initial_Call : Bool;   // Initial call of this OB
      Remanence : Bool;   // =True, if remanent data are available
   END_VAR
BEGIN

REGION Network 1
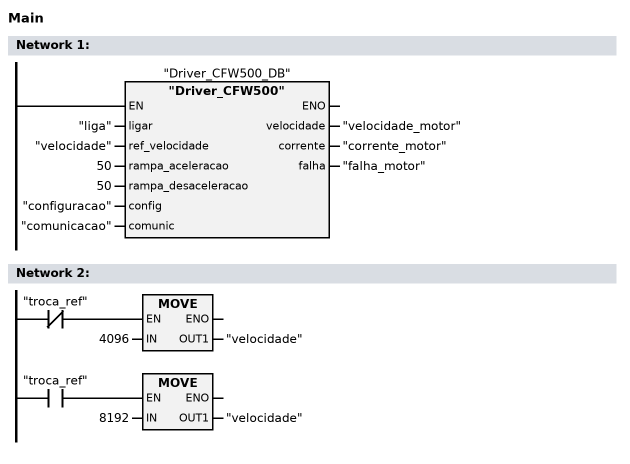
   RUNG wire#powerrail
      "Driver_CFW500_DB"(ligar := "liga", ref_velocidade := "velocidade", rampa_aceleracao := 50, rampa_desaceleracao := 50, config := "configuracao", comunic := "comunicacao", velocidade => "velocidade_motor", corrente => "corrente_motor", falha => "falha_motor")
   END_RUNG
   // the same network as SCL:
   "Driver_CFW500_DB"(ligar := "liga",   // "Driver_CFW500"
                      ref_velocidade := "velocidade",
                      rampa_aceleracao := 50,
                      rampa_desaceleracao := 50,
                      config := "configuracao",
                      comunic := "comunicacao",
                      velocidade => "velocidade_motor",
                      corrente => "corrente_motor",
                      falha => "falha_motor");
END_REGION

REGION Network 2
   RUNG wire#powerrail
      I_Contact( "troca_ref" )
      Move(in := 4096, out1 => "velocidade")
   END_RUNG
   RUNG wire#powerrail
      Contact( "troca_ref" )
      Move(in := 8192, out1 => "velocidade")
   END_RUNG
   // the same network as SCL:
   IF NOT "troca_ref" THEN "velocidade" := 4096; END_IF;
   IF "troca_ref" THEN "velocidade" := 8192; END_IF;
END_REGION
END_ORGANIZATION_BLOCK